FUNCTION "FC_Crt_PackArrived" : VOID
TITLE =%version: 0.17 %  CN: 32
//Function:
//Prepare and send message 'PackageReport' - Arrived
//
//History:
//This version  %created_by: nlhdl %
//              %date_created: maandag 6 juli 2015 10:31:50 %
//              %release: VI_CONV/RA_Dev_Oakham %
//
//Modification History:                                 By:      Date:     Rev:
//----------------------------------------------------  -------  --------  -----
//7324: ECS-P General from the RD to RA for platform    nlHdL    06-07-15   0.17
//23155: TIR in message for tubtrace                    nlHdL    24-04-15   0.17
//22147: Do not send package report arrived when PID=0  nlHdL    30-01-15   0.16
//22337: Remove the vibes1.x with the vibes 3.x         nlHdL    08-01-15   0.15
//19518: Block call update of FC_xxx_Record             nltny    07-08-14   0.06
//18032: package instr & package rep update             nlHdL    14-02-14   0.05
//17105: Messages sent with LNK instead of LIC          nlHdL    03-12-13   0.04
//15799: Block consistency update IO symbols, comment   nlHdL    23-09-13   0.03
//15170: Changed BTI to BTD for 4 digit Area num        nlHdL    13-08-13   0.02
//Initial Version based on version 0.10 ECS-P GEN       nlLvdG   31-05-13   0.01
//
FAMILY : VIBES
VERSION : 0.0


VAR_INPUT
  i_ID : DWORD ;	//ID Record HEX AAAA - ZZSS/OO.
  i_Data : INT ;	//Data needed to send the message
  i_FIFO_PLC_DB_num : INT ;	//Number of DB PLC FIFO
  i_DB_Event_Num : INT ;	//Number of DB event
END_VAR
VAR_TEMP
  t_AR1_Backup : DINT ;	//Save the contents of AR1
  t_Ret_Val_Word : WORD ;	//Return value Word, not used
  t_Ret_Val_Int : INT ;	//Return value Integer, not Used
  t_LIC : INT ;	//The LIC record used to create the message and send to SAC
  t_ECS : INT ;	//ECS record of LNK
  t_TIC_Number : INT ;	//TIC number
END_VAR
BEGIN
NETWORK
TITLE =AA: Store AR1 and Get Date and Time

      TAR1  ; // Store AR1
      T     #t_AR1_Backup;

      CALL "READ_CLK" (
           RET_VAL                  := #t_Ret_Val_Int,
           CDT                      := "DB_Outgoing_Msgs".PackageReport.body.EventTime);

NETWORK
TITLE =BA: Read ECS record

      CALL "FC_Read_Int_Record" (
           i_Record_Number          := #i_Data,
           i_P_INT_Record           := "DB_UDT_LNK_Record".ECS,
           i_DB                     := "DB_LNK_List",
           i_DB_Event_Num           := #i_DB_Event_Num,
           o_INT                    := #t_ECS);

      CALL "FC_Read_Int_Record" (
           i_Record_Number          := #i_Data,
           i_P_INT_Record           := "DB_UDT_LNK_Record".LIC,
           i_DB                     := "DB_LNK_List",
           i_DB_Event_Num           := #i_DB_Event_Num,
           o_INT                    := #t_LIC);

NETWORK
TITLE =CA: Write messageID

      AN    "M_Comm_Degraded"; // When in degraded mode
      JCN   CA01;

      L     211; // When NOT in degraded mode
      T     "DB_Outgoing_Msgs".PackageReport.body.MessageID;

      JU    CA99;

CA01: L     1211; // When in degraded mode
      T     "DB_Outgoing_Msgs".PackageReport.body.MessageID;

CA99: NOP   0;
NETWORK
TITLE =DA: Copy AreaID, ZoneID and SectionID

      L     #i_ID; // Load ID
      L     DW#16#FFFF0000; // Filter Area number only
      AD    ;
      SRD   16; // Slide Area nubmer to beginning AAAA0000 -> AAAA
      BTD   ; // Convert HEX to INT
      T     "DB_Outgoing_Msgs".PackageReport.body.AreaID; // Transfer to outgoing messages

      L     #i_ID; // Load ID
      L     DW#16#FF00; // Filter Zone number only
      AD    ;
      SRD   8; // Slide Zone nubmer to beginning 0000ZZ00 -> 0000ZZ
      BTI   ; // Convert HEX to INT
      T     "DB_Outgoing_Msgs".PackageReport.body.ZoneID; // Transfer to outgoing messages

      L     #i_ID; // Load ID
      L     DW#16#FF; // Filter Section number only
      AD    ;
      BTI   ; // Convert HEX to INT
      T     "DB_Outgoing_Msgs".PackageReport.body.EquipmentID; // Transfer to outgoing messages
NETWORK
TITLE =EA: Handle PIC code

      L     #t_LIC; // Write LIC number in the message
      T     "DB_Outgoing_Msgs".PackageReport.body.LIC;
NETWORK
TITLE =FA: Clear previous entries

      L     0;
      T     "DB_Outgoing_Msgs".PackageReport.body.ScreeningLevel.Process_1;
      T     "DB_Outgoing_Msgs".PackageReport.body.ScreeningLevel.Process_2;
      T     "DB_Outgoing_Msgs".PackageReport.body.ScreeningLevel.Process_3;
      T     "DB_Outgoing_Msgs".PackageReport.body.ScreeningLevel.Process_4;
      T     "DB_Outgoing_Msgs".PackageReport.body.ScreeningLevel.Process_5;
      T     "DB_Outgoing_Msgs".PackageReport.body.ScreeningResult.Process_1;
      T     "DB_Outgoing_Msgs".PackageReport.body.ScreeningResult.Process_2;
      T     "DB_Outgoing_Msgs".PackageReport.body.ScreeningResult.Process_3;
      T     "DB_Outgoing_Msgs".PackageReport.body.ScreeningResult.Process_4;
      T     "DB_Outgoing_Msgs".PackageReport.body.ScreeningResult.Process_5;

      L     '0';
      T     "DB_Outgoing_Msgs".PackageReport.body.ScanResult.LPN1[1];
      T     "DB_Outgoing_Msgs".PackageReport.body.ScanResult.LPN1[2];
      T     "DB_Outgoing_Msgs".PackageReport.body.ScanResult.LPN1[3];
      T     "DB_Outgoing_Msgs".PackageReport.body.ScanResult.LPN1[4];
      T     "DB_Outgoing_Msgs".PackageReport.body.ScanResult.LPN1[5];
      T     "DB_Outgoing_Msgs".PackageReport.body.ScanResult.LPN1[6];
      T     "DB_Outgoing_Msgs".PackageReport.body.ScanResult.LPN1[7];
      T     "DB_Outgoing_Msgs".PackageReport.body.ScanResult.LPN1[8];
      T     "DB_Outgoing_Msgs".PackageReport.body.ScanResult.LPN1[9];
      T     "DB_Outgoing_Msgs".PackageReport.body.ScanResult.LPN1[10];
      T     "DB_Outgoing_Msgs".PackageReport.body.ScanResult.LPN2[1];
      T     "DB_Outgoing_Msgs".PackageReport.body.ScanResult.LPN2[2];
      T     "DB_Outgoing_Msgs".PackageReport.body.ScanResult.LPN2[3];
      T     "DB_Outgoing_Msgs".PackageReport.body.ScanResult.LPN2[4];
      T     "DB_Outgoing_Msgs".PackageReport.body.ScanResult.LPN2[5];
      T     "DB_Outgoing_Msgs".PackageReport.body.ScanResult.LPN2[6];
      T     "DB_Outgoing_Msgs".PackageReport.body.ScanResult.LPN2[7];
      T     "DB_Outgoing_Msgs".PackageReport.body.ScanResult.LPN2[8];
      T     "DB_Outgoing_Msgs".PackageReport.body.ScanResult.LPN2[9];
      T     "DB_Outgoing_Msgs".PackageReport.body.ScanResult.LPN2[10];
      T     "DB_Outgoing_Msgs".PackageReport.body.ScanResult.LPN3[1];
      T     "DB_Outgoing_Msgs".PackageReport.body.ScanResult.LPN3[2];
      T     "DB_Outgoing_Msgs".PackageReport.body.ScanResult.LPN3[3];
      T     "DB_Outgoing_Msgs".PackageReport.body.ScanResult.LPN3[4];
      T     "DB_Outgoing_Msgs".PackageReport.body.ScanResult.LPN3[5];
      T     "DB_Outgoing_Msgs".PackageReport.body.ScanResult.LPN3[6];
      T     "DB_Outgoing_Msgs".PackageReport.body.ScanResult.LPN3[7];
      T     "DB_Outgoing_Msgs".PackageReport.body.ScanResult.LPN3[8];
      T     "DB_Outgoing_Msgs".PackageReport.body.ScanResult.LPN3[9];
      T     "DB_Outgoing_Msgs".PackageReport.body.ScanResult.LPN3[10];
      T     "DB_Outgoing_Msgs".PackageReport.body.ScreeningID[1];
      T     "DB_Outgoing_Msgs".PackageReport.body.ScreeningID[2];
      T     "DB_Outgoing_Msgs".PackageReport.body.ScreeningID[3];
      T     "DB_Outgoing_Msgs".PackageReport.body.ScreeningID[4];
      T     "DB_Outgoing_Msgs".PackageReport.body.ScreeningID[5];
      T     "DB_Outgoing_Msgs".PackageReport.body.ScreeningID[6];
      T     "DB_Outgoing_Msgs".PackageReport.body.ScreeningID[7];
      T     "DB_Outgoing_Msgs".PackageReport.body.ScreeningID[8];
      T     "DB_Outgoing_Msgs".PackageReport.body.ScreeningID[9];
      T     "DB_Outgoing_Msgs".PackageReport.body.ScreeningID[10];

NETWORK
TITLE =GA: Copy Information Record into message

      CALL "FC_Read_ANY_Record" (
           i_Record_Number          := #t_LIC,
           i_ANY_Data_Record        := "DB_UDT_LIC_Record".BIR,
           i_ANY_Data               := "DB_Outgoing_Msgs".PackageReport.body.BIR,
           i_DB                     := "DB_LIC_List",
           i_DB_Event_Num           := #i_DB_Event_Num);

      L     "DB_Outgoing_Msgs".PackageReport.body.BIR.PID;
      L     0;
      ==D   ;
      JCN   GA01;

      L     2209; // When PID = 0 then send log messagePackageReport no pid
      T     "DB_Outgoing_Msgs".PackageReport.body.MessageID;

GA01: NOP   0;
      L     0;
      T     "DB_Outgoing_Msgs".PackageReport.body.TIR.ID;

      L     "DB_Setting".common.External_Log_Level;
      L     4;
      >I    ;
      JCN   GA02;

      CALL "FC_Read_Int_Record" (
           i_Record_Number          := #i_Data,
           i_P_INT_Record           := "DB_UDT_LNK_Record".TIC,
           i_DB                     := "DB_LNK_List",
           i_DB_Event_Num           := #i_DB_Event_Num,
           o_INT                    := #t_TIC_Number);

      CALL "FC_Read_ANY_Record" (
           i_Record_Number          := #t_TIC_Number,
           i_ANY_Data_Record        := "DB_UDT_TIC_Record".TIR,
           i_ANY_Data               := "DB_Outgoing_Msgs".PackageReport.body.TIR,
           i_DB                     := "DB_TIC_List",
           i_DB_Event_Num           := #i_DB_Event_Num);

GA02: NOP   0;
NETWORK
TITLE =HA: Copy Arrived Location

      L     1; // 1= Arrived
      T     "DB_Outgoing_Msgs".PackageReport.body.Route_Result.Route_Result;

      CALL "FC_Read_Int_Record" (
           i_Record_Number          := #t_ECS,
           i_P_INT_Record           := "DB_UDT_ECS_Record".Routing_Result.Arrived_Location,
           i_DB                     := "DB_ECS_List",
           i_DB_Event_Num           := #i_DB_Event_Num,
           o_INT                    := "DB_Outgoing_Msgs".PackageReport.body.Route_Result.Location);
NETWORK
TITLE =IA: Put message in buffer

      CALL "BLKMOV" (
           SRCBLK                   := "DB_Outgoing_Msgs".Default,
           RET_VAL                  := #t_Ret_Val_Int,
           DSTBLK                   := "DB_Outgoing_Msgs".Merged_Message);

      CALL "BLKMOV" (
           SRCBLK                   := "DB_Outgoing_Msgs".PackageReport,
           RET_VAL                  := #t_Ret_Val_Int,
           DSTBLK                   := "DB_Outgoing_Msgs".Merged_Message);

      CALL "FC_FIFO" (
           i_FIFO_DB_Num            := #i_FIFO_PLC_DB_num,
           i_Mode                   := 'L',
           i_ANY_Data               := "DB_Outgoing_Msgs".Merged_Message,
           i_ID                     := #i_ID,
           o_RET_VAL_FIFO           := #t_Ret_Val_Word);

NETWORK
TITLE =JA: Restore AR1

      L     #t_AR1_Backup;
      LAR1  ;
END_FUNCTION

